KUKA KRL program: adjust_changes.src, Adjust_Changes.dat

--- adjust_changes.src ---
&ACCESS RVO1
&REL 57
&PARAM EDITMASK = *
&PARAM TEMPLATE = C:\KRC\Roboter\Template\vorgabe
&PARAM DISKPATH = KRC:\R1\Program\Production
DEF Adjust_Changes( )
   ;FOLD INI;%{PE}
      ;FOLD BASISTECH INI
         GLOBAL INTERRUPT DECL 3 WHEN $STOPMESS==TRUE DO IR_STOPM ( )
         INTERRUPT ON 3
         BAS (#INITMOV,0 )
      ;ENDFOLD (BASISTECH INI)
      ;FOLD USER INI
         ;Make your modifications here

      ;ENDFOLD (USER INI)
   ;ENDFOLD (INI)

   Xdummy_point = $POS_ACT
   PTP Xdummy_point

   ;FOLD HandShake[24 : Adjust changes], WAIT on Response
      HandShake_Set (24,false)
      HandShake_Check (24,false)
   ;ENDFOLD

   Xdummy_point = $POS_ACT
   PTP Xdummy_point

   WHILE doneAdjusting == FALSE
      BARRELPOSAUX = $NULLFRAME
      jogDone = false
      WAIT SEC 0.1

      ; FOLD INI Jog Up Down Override
         IF jogUPSEAM  THEN
            BARRELPOSAUX.x = 0.05
            jogDone = true
         ENDIF

         IF jogDOWNSEAM   THEN
            BARRELPOSAUX.x = -0.05
            jogDone = true
         ENDIF

      ; ENDFOLD INI

      ; FOLD INI Jog In Out Override
         IF goIn  THEN
            BARRELPOSAUX.Z = 0.05
            jogDone = true
         ENDIF

         IF goOut  THEN
            BARRELPOSAUX.Z = -0.05
            jogDone = true
         ENDIF

         IF jogDone THEN
          ; Adjust
         LIN_REL BARRELPOSAUX #TOOL
         ENDIF

   ENDWHILE
   Xdummy_point = $POS_ACT
   PTP Xdummy_point
   Exit_Program()

END

--- Adjust_Changes.dat ---
&ACCESS RVO1
&REL 57
&PARAM EDITMASK = *
&PARAM TEMPLATE = C:\KRC\Roboter\Template\vorgabe
&PARAM DISKPATH = KRC:\R1\Program\Production
DEFDAT  Adjust_Changes
;FOLD EXTERNAL DECLARATIONS;%{PE}%MKUKATPBASIS,%CEXT,%VCOMMON,%P
;FOLD BASISTECH EXT;%{PE}%MKUKATPBASIS,%CEXT,%VEXT,%P
EXT  BAS (BAS_COMMAND  :IN,REAL  :IN )
;ENDFOLD (BASISTECH EXT)
;FOLD USER EXT;%{E}%MKUKATPUSER,%CEXT,%VEXT,%P
;Make your modifications here
;ENDFOLD (USER EXT)
;ENDFOLD (EXTERNAL DECLARATIONS)

DECL BOOL throwawaybool
DECL REAL barrel60inch = -300.0
DECL REAL barrel72ich = 7.0

 DECL int nType

DECL FDAT FHOME2={TOOL_NO 1,BASE_NO 0,IPO_FRAME #BASE,POINT2[] " "}
DECL PDAT PPDAT1={VEL 1.0000,ACC 5.00000,APO_DIST 100.000,APO_MODE #CDIS,GEAR_JERK 50.0000,EXAX_IGN 0}

ENDDAT
